(* Logix 5000 project; controller SPECK Emulate 5570 rev 30.12; software revision 30.00 *)

TASK MainTask (periodic, rate 5000 ms, priority 1, watchdog 5000 ms) : MainProgram

MODULES
   Local : Emulate 5570 (ICP 2, rev 30.12)
       : vendor 1 type 0 code 15 (ICP 0, rev 1.1, Output RPI 50 ms)
END_MODULES

TYPE UDT_BA :
STRUCT
   AL : BOOL;
END_STRUCT
END_TYPE

PROGRAM MainProgram   (* main routine MainRoutine *)
VAR
   SCAN_CYCLE_TIME : DINT;
   Speck_AS_res : DINT[2];
   Speck_AS_tmp : DINT;
   Speck_AS_X : DINT[2] := ([0] := -536870912);
   Speck_AS_Y : DINT[2] := ([0] := 1610612736);
   Speck_Block_size : DINT;
   Speck_Carry_Bit : DINT;
   Speck_Ciphertext : DINT[2,2];
   Speck_dec_i : DINT;
   Speck_dec_j : DINT;
   Speck_enc_i : DINT;
   Speck_enc_j : DINT;
   Speck_i : DINT;
   Speck_j : DINT;
   Speck_key_size : DINT;
   Speck_Plaintext : DINT[2,2];
   Speck_Rd_Max : DINT;
   Speck_Rotate_Result : DINT[2];
   Speck_Round_Keys : DINT[34,2];
   Speck_Sign_Bits : DINT[2];
   Speck_SR_m : DINT[2];
   Speck_tmp : DINT;
   Speck_tmp1 : DINT;
   Speck_Ver : DINT;
   Speck_x : DINT[2];
   Speck_y : DINT[2];
END_VAR

ROUTINE MainRoutine   (* ladder *)
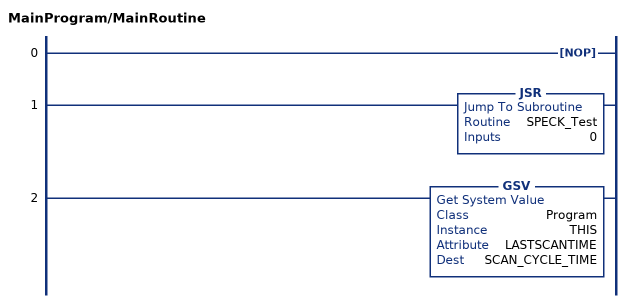
   0: NOP();
   1: JSR(SPECK_Test,0);
   2: GSV(Program,THIS,LASTSCANTIME,SCAN_CYCLE_TIME);
END_ROUTINE

ROUTINE SPECK_Add   (* structured text *)
   	//big addition low 32-bit
   		Speck_AS_res[0]:=0;
   		Speck_AS_res[1]:=0;
   		Speck_Sign_Bits[0].[0]:= Speck_AS_X[0].30; //keep the sign bit for big addition
   		Speck_Sign_Bits[0].[1]:= Speck_AS_X[0].31;
   		Speck_AS_X[0].31:=0;
   		Speck_AS_X[0].30:=0;
   
   		Speck_Sign_Bits[1].[0]:= Speck_AS_Y[0].30; //keep the sign bit for big addition
   		Speck_Sign_Bits[1].[1]:= Speck_AS_Y[0].31;
   		Speck_AS_Y[0].31:=0;
   		Speck_AS_Y[0].30:=0;
   
   		Speck_AS_res[0] := Speck_AS_X[0]+Speck_AS_Y[0];
   
   		Speck_Carry_Bit.[0]:= Speck_AS_res[0].30;
   
   		Speck_AS_tmp:=Speck_Sign_Bits[1]+Speck_Sign_Bits[0]+Speck_Carry_Bit;
   
   		Speck_AS_res[0].[30]:= Speck_AS_tmp.[0];
   		Speck_AS_res[0].[31]:= Speck_AS_tmp.[1];
   
   		Speck_Carry_Bit.[0]:= Speck_AS_tmp.[2];
   
   
   		Speck_AS_tmp:=0;
   		Speck_Sign_Bits[0]:=0;
   		Speck_Sign_Bits[1]:=0;
   
   //add high 32-bit
   if Speck_Ver>2 then
   		Speck_Sign_Bits[0].[0]:= Speck_AS_X[1].30; //keep the sign bit for big addition
   		Speck_Sign_Bits[0].[1]:= Speck_AS_X[1].31;
   		Speck_AS_X[1].31:=0;
   		Speck_AS_X[1].30:=0;
   
   		Speck_Sign_Bits[1].[0]:= Speck_AS_Y[1].30; //keep the sign bit for big addition
   		Speck_Sign_Bits[1].[1]:= Speck_AS_Y[1].31;
   		Speck_AS_Y[1].31:=0;
   		Speck_AS_Y[1].30:=0;
   
   		Speck_AS_res[1]:=Speck_AS_X[1]+Speck_AS_Y[1]+Speck_Carry_Bit;
   
   		Speck_Carry_Bit.[0]:= Speck_AS_res[1].30;
   
   		Speck_AS_tmp:=Speck_Sign_Bits[1]+Speck_Sign_Bits[0]+Speck_Carry_Bit;
   
   		Speck_AS_res[1].[30]:= Speck_AS_tmp.[0];
   		Speck_AS_res[1].[31]:= Speck_AS_tmp.[1];
   end_if;
   
   		//clear
   		Speck_Carry_Bit:=0;
   		Speck_AS_tmp:=0;
   		Speck_Sign_Bits[0]:=0;
   		Speck_Sign_Bits[1]:=0;
   		Speck_AS_X[0]:=0;
   		Speck_AS_X[1]:=0;
   		Speck_AS_Y[0]:=0;
   		Speck_AS_Y[1]:=0;
   
   
END_ROUTINE

ROUTINE SPECK_ClearKey   (* structured text *)
   
   Speck_Round_Keys[0,0]:=0;
   Speck_Round_Keys[1,0]:=0;
   Speck_Round_Keys[2,0]:=0;
   Speck_Round_Keys[3,0]:=0;
   Speck_Round_Keys[4,0]:=0;
   Speck_Round_Keys[5,0]:=0;
   Speck_Round_Keys[6,0]:=0;
   Speck_Round_Keys[7,0]:=0;
   Speck_Round_Keys[8,0]:=0;
   Speck_Round_Keys[9,0]:=0;
   Speck_Round_Keys[10,0]:=0;
   Speck_Round_Keys[11,0]:=0;
   Speck_Round_Keys[12,0]:=0;
   Speck_Round_Keys[13,0]:=0;
   Speck_Round_Keys[14,0]:=0;
   Speck_Round_Keys[15,0]:=0;
   Speck_Round_Keys[16,0]:=0;
   Speck_Round_Keys[17,0]:=0;
   Speck_Round_Keys[18,0]:=0;
   Speck_Round_Keys[19,0]:=0;
   Speck_Round_Keys[20,0]:=0;
   Speck_Round_Keys[21,0]:=0;
   Speck_Round_Keys[22,0]:=0;
   Speck_Round_Keys[23,0]:=0;
   Speck_Round_Keys[24,0]:=0;
   Speck_Round_Keys[25,0]:=0;
   Speck_Round_Keys[26,0]:=0;
END_ROUTINE

ROUTINE SPECK_Dec   (* structured text *)
   
   JSR(SPECK_Init);
   
   
   
   
   Case Speck_Ver Of
   
   0,1,2:
   	Speck_Plaintext[0,0]:=Speck_Ciphertext[0,0];
   	Speck_Plaintext[1,0]:=Speck_Ciphertext[1,0];
   
   	For Speck_i:=Speck_Rd_Max to 0 by -1 do
   
   		Speck_AS_res[0]:= Speck_Plaintext[1,0] XOR Speck_Plaintext[0,0];
   
   		Speck_SR_m[0]:=Speck_AS_res[0];
   		JSR(SPECK_Rotate_Right_Dec);      //rotate based on Speck_AS_res[0]
   
   		Speck_Plaintext[0,0]:= Speck_Rotate_Result[0];
   
   		Speck_AS_X[0]:= Speck_Plaintext[1,0] XOR Speck_Round_Keys[Speck_i,0];
   
   
   
   		if Speck_Ver=0 Then
   			Speck_AS_X[0].16:=1;
   			Speck_AS_res[0]:= (Speck_AS_X[0]- Speck_Plaintext[0,0]) AND 16#0000ffff; //??AND 16#ffff;
   		Else
   			Speck_AS_Y[0]:=Speck_Plaintext[0,0];
   			JSR(SPECK_Sub);
   		End_if;
   		Speck_SR_m[0]:=Speck_AS_res[0];
   		JSR(SPECK_Rotate_Left_Dec);      //rotate based on Speck_AS_res[0]
   		Speck_Plaintext[1,0]:=Speck_Rotate_Result[0];
   
   	End_for;
   
   3,4,5:
   	Speck_Plaintext[0,0]:=Speck_Ciphertext[0,0];
   	Speck_Plaintext[0,1]:=Speck_Ciphertext[0,1];
   	Speck_Plaintext[1,0]:=Speck_Ciphertext[1,0];
   	Speck_Plaintext[1,1]:=Speck_Ciphertext[1,1];
   
   	For Speck_i:=Speck_Rd_Max to 0 by -1 do
   
   		Speck_AS_res[0]:= Speck_Plaintext[0,0] XOR Speck_Plaintext[1,0];
   		Speck_AS_res[1]:= Speck_Plaintext[0,1] XOR Speck_Plaintext[1,1];
   
   
   		Speck_SR_m[0]:=Speck_AS_res[0];
   		Speck_SR_m[1]:=Speck_AS_res[1];
   		JSR(SPECK_Rotate_Right_Dec);      //rotate based on Speck_AS_res[0] and Speck_AS_res[1]
   
   		Speck_Plaintext[0,0]:= Speck_Rotate_Result[0];
   		Speck_Plaintext[0,1]:= Speck_Rotate_Result[1];
   
   		Speck_AS_X[0]:= Speck_Plaintext[1,0] XOR Speck_Round_Keys[Speck_i,0];
   		Speck_AS_X[1]:= Speck_Plaintext[1,1] XOR Speck_Round_Keys[Speck_i,1];
   
   
   		Speck_AS_Y[0]:=Speck_Plaintext[0,0];
   		Speck_AS_Y[1]:=Speck_Plaintext[0,1];
   		JSR(SPECK_Sub);
   
   		Speck_SR_m[0]:=Speck_AS_res[0];
   		Speck_SR_m[1]:=Speck_AS_res[1];
   		JSR(SPECK_Rotate_Left_Dec);      //rotate based on Speck_AS_res[0] and Speck_AS_res[1]
   		Speck_Plaintext[1,0]:=Speck_Rotate_Result[0];
   		Speck_Plaintext[1,1]:=Speck_Rotate_Result[1];
   	End_for;
   
   End_Case;
   
   
   
   
   
   
   JSR(SPECK_ClearKey);
   
   
   
   
   
   
   
   
END_ROUTINE

ROUTINE SPECK_Enc   (* structured text *)
   
   JSR(SPECK_Init);
   
   
   Case Speck_Ver Of
   
   0,1,2:
   	Speck_Ciphertext[0,0]:=Speck_Plaintext[0,0];
   	Speck_Ciphertext[1,0]:=Speck_Plaintext[1,0];
   
   	For Speck_i:=0 to Speck_Rd_Max by 1 do
   		Speck_SR_m[0]:=Speck_Ciphertext[1,0];
   		JSR(SPECK_Rotate_Right_Enc);       //c1>>>>
   
   		if Speck_Ver=0 Then
   			Speck_Ciphertext[1,0]:= (Speck_Rotate_Result[0] + Speck_Ciphertext[0,0]) XOR Speck_Round_Keys[Speck_i,0];
   			Speck_Ciphertext[1,0]:= Speck_Ciphertext[1,0] AND 16#0000ffff;
   		Else
   			Speck_AS_X[0]:=Speck_Rotate_Result[0];
   			Speck_AS_Y[0]:=Speck_Ciphertext[0,0];
   			JSR(SPECK_Add);
   			Speck_Ciphertext[1,0]:= Speck_AS_res[0] XOR Speck_Round_Keys[Speck_i,0];
   		End_if;
   
   
   		Speck_SR_m[0]:=Speck_Ciphertext[0,0];
   		JSR(SPECK_Rotate_Left_Enc);   //p0<<<
   		Speck_Ciphertext[0,0]:=Speck_Rotate_Result[0] XOR Speck_Ciphertext[1,0];
   	End_for;
   
   3,4,5:
   	Speck_Ciphertext[0,0]:=Speck_Plaintext[0,0];
   	Speck_Ciphertext[0,1]:=Speck_Plaintext[0,1];
   	Speck_Ciphertext[1,0]:=Speck_Plaintext[1,0];
   	Speck_Ciphertext[1,1]:=Speck_Plaintext[1,1];
   
   	For Speck_i:=0 to Speck_Rd_Max by 1 do
   		Speck_SR_m[0]:=Speck_Ciphertext[1,0];
   		Speck_SR_m[1]:=Speck_Ciphertext[1,1];
   		JSR(SPECK_Rotate_Right_Enc);       //c1>>>>
   
   		Speck_AS_X[0]:=Speck_Rotate_Result[0];
   		Speck_AS_X[1]:=Speck_Rotate_Result[1];
   		Speck_AS_Y[0]:=Speck_Ciphertext[0,0];
   		Speck_AS_Y[1]:=Speck_Ciphertext[0,1];
   		JSR(SPECK_Add);
   		Speck_Ciphertext[1,0]:= Speck_AS_res[0] XOR Speck_Round_Keys[Speck_i,0];
   	 	Speck_Ciphertext[1,1]:= Speck_AS_res[1] XOR Speck_Round_Keys[Speck_i,1];
   
   		Speck_SR_m[0]:=Speck_Ciphertext[0,0];
   		Speck_SR_m[1]:=Speck_Ciphertext[0,1];
   		JSR(SPECK_Rotate_Left_Enc);   //c0<<<
   		Speck_Ciphertext[0,0]:=Speck_Rotate_Result[0] XOR Speck_Ciphertext[1,0];
   		Speck_Ciphertext[0,1]:=Speck_Rotate_Result[1] XOR Speck_Ciphertext[1,1];
   	End_for;
   
   End_Case;
   
   
   JSR(SPECK_ClearKey);
   
   
   
   
   
   
END_ROUTINE

ROUTINE SPECK_Init   (* structured text *)
   CASE Speck_Ver Of
   	0:
   		//Speck_Rd_Max:=21;
   		Speck_Rd_Max:=21;
   		Speck_Round_Keys[0,0]:=256;
   		Speck_Round_Keys[1,0]:=5394;
   		Speck_Round_Keys[2,0]:=24957;
   		Speck_Round_Keys[3,0]:=5208;
   		Speck_Round_Keys[4,0]:=26905;
   		Speck_Round_Keys[5,0]:=30690;
   		Speck_Round_Keys[6,0]:=3209;
   		Speck_Round_Keys[7,0]:=52443;
   		Speck_Round_Keys[8,0]:=61418;
   		Speck_Round_Keys[9,0]:=20019;
   		Speck_Round_Keys[10,0]:=30452;
   		Speck_Round_Keys[11,0]:=22902;
   		Speck_Round_Keys[12,0]:=61067;
   		Speck_Round_Keys[13,0]:=56068;
   		Speck_Round_Keys[14,0]:=17943;
   		Speck_Round_Keys[15,0]:=62334;
   		Speck_Round_Keys[16,0]:=34740;
   		Speck_Round_Keys[17,0]:=36554;
   		Speck_Round_Keys[18,0]:=60827;
   		Speck_Round_Keys[19,0]:=14930;
   		Speck_Round_Keys[20,0]:=33321;
   		Speck_Round_Keys[21,0]:=60772;
   
   	1:
   		Speck_Rd_Max:=25;
   		Speck_Round_Keys[0,0]:=50462976;
   		Speck_Round_Keys[1,0]:=320668425;
   		Speck_Round_Keys[2,0]:=-1143468717;
   		Speck_Round_Keys[3,0]:=438530241;
   		Speck_Round_Keys[4,0]:=-463657251;
   		Speck_Round_Keys[5,0]:=1674264348;
   		Speck_Round_Keys[6,0]:=660176218;
   		Speck_Round_Keys[7,0]:=542209460;
   		Speck_Round_Keys[8,0]:=-620635233;
   		Speck_Round_Keys[9,0]:=-1743607096;
   		Speck_Round_Keys[10,0]:=377054067;
   		Speck_Round_Keys[11,0]:=-9280389;
   		Speck_Round_Keys[12,0]:=-858098844;
   		Speck_Round_Keys[13,0]:=-688605239;
   		Speck_Round_Keys[14,0]:=629784410;
   		Speck_Round_Keys[15,0]:=963910745;
   		Speck_Round_Keys[16,0]:=-2052674916;
   		Speck_Round_Keys[17,0]:=546222198;
   		Speck_Round_Keys[18,0]:=1906914590;
   		Speck_Round_Keys[19,0]:=-1895867933;
   		Speck_Round_Keys[20,0]:=1234172310;
   		Speck_Round_Keys[21,0]:=367819809;
   		Speck_Round_Keys[22,0]:=256446538;
   		Speck_Round_Keys[23,0]:=-655744580;
   		Speck_Round_Keys[24,0]:=-589610660;
   		Speck_Round_Keys[25,0]:=799533313;
   
   	2:
   		Speck_Rd_Max:=26;
   		Speck_Round_Keys[0,0]:=50462976;
   		Speck_Round_Keys[1,0]:=320668425;
   		Speck_Round_Keys[2,0]:=-1143468717;
   		Speck_Round_Keys[3,0]:=1696098252;
   		Speck_Round_Keys[4,0]:=1189104311;
   		Speck_Round_Keys[5,0]:=1426141042;
   		Speck_Round_Keys[6,0]:=246709480;
   		Speck_Round_Keys[7,0]:=-1769912550;
   		Speck_Round_Keys[8,0]:=-353799609;
   		Speck_Round_Keys[9,0]:=853261689;
   		Speck_Round_Keys[10,0]:=459475929;
   		Speck_Round_Keys[11,0]:=1977201121;
   		Speck_Round_Keys[12,0]:=317902096;
   		Speck_Round_Keys[13,0]:=-1273568388;
   		Speck_Round_Keys[14,0]:=2104671875;
   		Speck_Round_Keys[15,0]:=1924860368;
   		Speck_Round_Keys[16,0]:=-83442473;
   		Speck_Round_Keys[17,0]:=-1177375533;
   		Speck_Round_Keys[18,0]:=1274985820;
   		Speck_Round_Keys[19,0]:=-6786794;
   		Speck_Round_Keys[20,0]:=-1757815548;
   		Speck_Round_Keys[21,0]:=-512646929;
   		Speck_Round_Keys[22,0]:=-576779808;
   		Speck_Round_Keys[23,0]:=2113096485;
   		Speck_Round_Keys[24,0]:=-1495903407;
   		Speck_Round_Keys[25,0]:=1881079754;
   		Speck_Round_Keys[26,0]:=323482756;
   	3:
   		Speck_Rd_Max:=31;
   		Speck_Round_Keys[0,0]:=50462976;
   		Speck_Round_Keys[0,1]:=117835012;
   		Speck_Round_Keys[1,0]:=387777289;
   		Speck_Round_Keys[1,1]:=925186865;
   		Speck_Round_Keys[2,0]:=-1866200996;
   		Speck_Round_Keys[2,1]:=-115504692;
   		Speck_Round_Keys[3,0]:=1389131401;
   		Speck_Round_Keys[3,1]:=-961417096;
   		Speck_Round_Keys[4,0]:=-104671504;
   		Speck_Round_Keys[4,1]:=22007284;
   		Speck_Round_Keys[5,0]:=-31141930;
   		Speck_Round_Keys[5,1]:=-1241849372;
   		Speck_Round_Keys[6,0]:=-1334608642;
   		Speck_Round_Keys[6,1]:=-1553110700;
   		Speck_Round_Keys[7,0]:=-1607518733;
   		Speck_Round_Keys[7,1]:=-183408354;
   		Speck_Round_Keys[8,0]:=1512785245;
   		Speck_Round_Keys[8,1]:=1400155063;
   		Speck_Round_Keys[9,0]:=1306309285;
   		Speck_Round_Keys[9,1]:=-1915357664;
   		Speck_Round_Keys[10,0]:=-2036552680;
   		Speck_Round_Keys[10,1]:=-1304176695;
   		Speck_Round_Keys[11,0]:=1717585310;
   		Speck_Round_Keys[11,1]:=1967028860;
   		Speck_Round_Keys[12,0]:=-1515133381;
   		Speck_Round_Keys[12,1]:=2027309219;
   		Speck_Round_Keys[13,0]:=-876566318;
   		Speck_Round_Keys[13,1]:=-2028655837;
   		Speck_Round_Keys[14,0]:=1420015346;
   		Speck_Round_Keys[14,1]:=-1459647604;
   		Speck_Round_Keys[15,0]:=1135864441;
   		Speck_Round_Keys[15,1]:=1215544892;
   		Speck_Round_Keys[16,0]:=-1090139373;
   		Speck_Round_Keys[16,1]:=1998503932;
   		Speck_Round_Keys[17,0]:=629554464;
   		Speck_Round_Keys[17,1]:=-391725905;
   		Speck_Round_Keys[18,0]:=1548881043;
   		Speck_Round_Keys[18,1]:=-423433589;
   		Speck_Round_Keys[19,0]:=-1403906827;
   		Speck_Round_Keys[19,1]:=1299297729;
   		Speck_Round_Keys[20,0]:=623931612;
   		Speck_Round_Keys[20,1]:=-597642578;
   		Speck_Round_Keys[21,0]:=-503605439;
   		Speck_Round_Keys[21,1]:=-1340273989;
   		Speck_Round_Keys[22,0]:=-1558661814;
   		Speck_Round_Keys[22,1]:=-677874044;
   		Speck_Round_Keys[23,0]:=-436153575;
   		Speck_Round_Keys[23,1]:=-1574153598;
   		Speck_Round_Keys[24,0]:=-1107754936;
   		Speck_Round_Keys[24,1]:=-534129026;
   		Speck_Round_Keys[25,0]:=-934347329;
   		Speck_Round_Keys[25,1]:=1733661236;
   		Speck_Round_Keys[26,0]:=-889099940;
   		Speck_Round_Keys[26,1]:=1696021744;
   		Speck_Round_Keys[27,0]:=2038535449;
   		Speck_Round_Keys[27,1]:=617553688;
   		Speck_Round_Keys[28,0]:=-609241302;
   		Speck_Round_Keys[28,1]:=950234834;
   		Speck_Round_Keys[29,0]:=834331396;
   		Speck_Round_Keys[29,1]:=-556188418;
   		Speck_Round_Keys[30,0]:=393261669;
   		Speck_Round_Keys[30,1]:=-985851719;
   		Speck_Round_Keys[31,0]:=-611399361;
   		Speck_Round_Keys[31,1]:=563726448;
   
   	4:
   		Speck_Rd_Max:=32;
   		Speck_Round_Keys[0,0]:=50462976;
   		Speck_Round_Keys[0,1]:=117835012;
   		Speck_Round_Keys[1,0]:=387777289;
   		Speck_Round_Keys[1,1]:=925186865;
   		Speck_Round_Keys[2,0]:=-1814557358;
   		Speck_Round_Keys[2,1]:=-32143154;
   		Speck_Round_Keys[3,0]:=975663304;
   		Speck_Round_Keys[3,1]:=-142025835;
   		Speck_Round_Keys[4,0]:=1365845657;
   		Speck_Round_Keys[4,1]:=-1365849265;
   		Speck_Round_Keys[5,0]:=-1203291782;
   		Speck_Round_Keys[5,1]:=2032907671;
   		Speck_Round_Keys[6,0]:=1560168396;
   		Speck_Round_Keys[6,1]:=-1637668590;
   		Speck_Round_Keys[7,0]:=-1379701829;
   		Speck_Round_Keys[7,1]:=-1503031408;
   		Speck_Round_Keys[8,0]:=863596189;
   		Speck_Round_Keys[8,1]:=-158551405;
   		Speck_Round_Keys[9,0]:=-1375147243;
   		Speck_Round_Keys[9,1]:=1636284355;
   		Speck_Round_Keys[10,0]:=-1272900118;
   		Speck_Round_Keys[10,1]:=-1368340852;
   		Speck_Round_Keys[11,0]:=-1352763690;
   		Speck_Round_Keys[11,1]:=-624911147;
   		Speck_Round_Keys[12,0]:=1003580318;
   		Speck_Round_Keys[12,1]:=-899281693;
   		Speck_Round_Keys[13,0]:=894738061;
   		Speck_Round_Keys[13,1]:=490681490;
   		Speck_Round_Keys[14,0]:=691090703;
   		Speck_Round_Keys[14,1]:=-1398656019;
   		Speck_Round_Keys[15,0]:=-57361246;
   		Speck_Round_Keys[15,1]:=1122098217;
   		Speck_Round_Keys[16,0]:=-1648511106;
   		Speck_Round_Keys[16,1]:=-1121331570;
   		Speck_Round_Keys[17,0]:=866086775;
   		Speck_Round_Keys[17,1]:=1964995237;
   		Speck_Round_Keys[18,0]:=1776548963;
   		Speck_Round_Keys[18,1]:=1228016885;
   		Speck_Round_Keys[19,0]:=1960676415;
   		Speck_Round_Keys[19,1]:=-2107754217;
   		Speck_Round_Keys[20,0]:=-146881239;
   		Speck_Round_Keys[20,1]:=1236388362;
   		Speck_Round_Keys[21,0]:=176991942;
   		Speck_Round_Keys[21,1]:=586401854;
   		Speck_Round_Keys[22,0]:=-272894130;
   		Speck_Round_Keys[22,1]:=-271496784;
   		Speck_Round_Keys[23,0]:=615566260;
   		Speck_Round_Keys[23,1]:=46828238;
   		Speck_Round_Keys[24,0]:=1089140610;
   		Speck_Round_Keys[24,1]:=-1802072153;
   		Speck_Round_Keys[25,0]:=-1928078593;
   		Speck_Round_Keys[25,1]:=-56185516;
   		Speck_Round_Keys[26,0]:=199725135;
   		Speck_Round_Keys[26,1]:=-98821494;
   		Speck_Round_Keys[27,0]:=625825488;
   		Speck_Round_Keys[27,1]:=898955530;
   		Speck_Round_Keys[28,0]:=2044356237;
   		Speck_Round_Keys[28,1]:=1226041899;
   		Speck_Round_Keys[29,0]:=445115415;
   		Speck_Round_Keys[29,1]:=-1335488765;
   		Speck_Round_Keys[30,0]:=1088748615;
   		Speck_Round_Keys[30,1]:=1048296253;
   		Speck_Round_Keys[31,0]:=-1633766600;
   		Speck_Round_Keys[31,1]:=1336503665;
   		Speck_Round_Keys[32,0]:=818288393;
   		Speck_Round_Keys[32,1]:=925749944;
   
   	5:
   		Speck_Rd_Max:=33;
   		Speck_Round_Keys[0,0]:=50462976;
   		Speck_Round_Keys[0,1]:=117835012;
   		Speck_Round_Keys[1,0]:=387777289;
   		Speck_Round_Keys[1,1]:=925186865;
   		Speck_Round_Keys[2,0]:=-1814557358;
   		Speck_Round_Keys[2,1]:=-32143154;
   		Speck_Round_Keys[3,0]:=825445886;
   		Speck_Round_Keys[3,1]:=-426188641;
   		Speck_Round_Keys[4,0]:=-875023107;
   		Speck_Round_Keys[4,1]:=-614403765;
   		Speck_Round_Keys[5,0]:=1287832312;
   		Speck_Round_Keys[5,1]:=766486467;
   		Speck_Round_Keys[6,0]:=1583653339;
   		Speck_Round_Keys[6,1]:=-71769488;
   		Speck_Round_Keys[7,0]:=-477893905;
   		Speck_Round_Keys[7,1]:=-613443100;
   		Speck_Round_Keys[8,0]:=-1668630227;
   		Speck_Round_Keys[8,1]:=689605941;
   		Speck_Round_Keys[9,0]:=-493428094;
   		Speck_Round_Keys[9,1]:=191183550;
   		Speck_Round_Keys[10,0]:=1544592767;
   		Speck_Round_Keys[10,1]:=1614952126;
   		Speck_Round_Keys[11,0]:=-1911170916;
   		Speck_Round_Keys[11,1]:=-1239078670;
   		Speck_Round_Keys[12,0]:=-793616599;
   		Speck_Round_Keys[12,1]:=272735697;
   		Speck_Round_Keys[13,0]:=-1670774794;
   		Speck_Round_Keys[13,1]:=-42866885;
   		Speck_Round_Keys[14,0]:=2140630675;
   		Speck_Round_Keys[14,1]:=-1901518332;
   		Speck_Round_Keys[15,0]:=965541820;
   		Speck_Round_Keys[15,1]:=771988221;
   		Speck_Round_Keys[16,0]:=583075628;
   		Speck_Round_Keys[16,1]:=-1667248145;
   		Speck_Round_Keys[17,0]:=-313137463;
   		Speck_Round_Keys[17,1]:=637176179;
   		Speck_Round_Keys[18,0]:=-1498142708;
   		Speck_Round_Keys[18,1]:=1770100833;
   		Speck_Round_Keys[19,0]:=-1744597129;
   		Speck_Round_Keys[19,1]:=2070075508;
   		Speck_Round_Keys[20,0]:=1659016958;
   		Speck_Round_Keys[20,1]:=-231399730;
   		Speck_Round_Keys[21,0]:=1991902719;
   		Speck_Round_Keys[21,1]:=-1496087855;
   		Speck_Round_Keys[22,0]:=1169655590;
   		Speck_Round_Keys[22,1]:=-1919490457;
   		Speck_Round_Keys[23,0]:=-1645822159;
   		Speck_Round_Keys[23,1]:=-1099482754;
   		Speck_Round_Keys[24,0]:=-1350724487;
   		Speck_Round_Keys[24,1]:=890732295;
   		Speck_Round_Keys[25,0]:=-410951696;
   		Speck_Round_Keys[25,1]:=-1201049147;
   		Speck_Round_Keys[26,0]:=272319978;
   		Speck_Round_Keys[26,1]:=2104999935;
   		Speck_Round_Keys[27,0]:=-2103336674;
   		Speck_Round_Keys[27,1]:=-1719430836;
   		Speck_Round_Keys[28,0]:=1848838133;
   		Speck_Round_Keys[28,1]:=512289202;
   		Speck_Round_Keys[29,0]:=1338443291;
   		Speck_Round_Keys[29,1]:=2046847095;
   		Speck_Round_Keys[30,0]:=2113057135;
   		Speck_Round_Keys[30,1]:=393340252;
   		Speck_Round_Keys[31,0]:=-1141349352;
   		Speck_Round_Keys[31,1]:=-1563733213;
   		Speck_Round_Keys[32,0]:=2146821003;
   		Speck_Round_Keys[32,1]:=1073939284;
   		Speck_Round_Keys[33,0]:=-1705594250;
   		Speck_Round_Keys[33,1]:=-187535528;
   End_CASE;
   
END_ROUTINE

ROUTINE SPECK_Rotate_Left_Dec   (* structured text *)
   Speck_Rotate_Result[0]:=0;
   Speck_Rotate_Result[1]:=0;
   
   CASE Speck_Ver Of
   	0:
   		Speck_Rotate_Result[0].[6]:=Speck_SR_m[0].[15];
   		Speck_Rotate_Result[0].[5]:=Speck_SR_m[0].[14];
   		Speck_Rotate_Result[0].[4]:=Speck_SR_m[0].[13];
   		Speck_Rotate_Result[0].[3]:=Speck_SR_m[0].[12];
   		Speck_Rotate_Result[0].[2]:=Speck_SR_m[0].[11];
   		Speck_Rotate_Result[0].[1]:=Speck_SR_m[0].[10];
   		Speck_Rotate_Result[0].[0]:=Speck_SR_m[0].[9];
   		Speck_Rotate_Result[0].[15]:=Speck_SR_m[0].[8];
   		Speck_Rotate_Result[0].[14]:=Speck_SR_m[0].[7];
   		Speck_Rotate_Result[0].[13]:=Speck_SR_m[0].[6];
   		Speck_Rotate_Result[0].[12]:=Speck_SR_m[0].[5];
   		Speck_Rotate_Result[0].[11]:=Speck_SR_m[0].[4];
   		Speck_Rotate_Result[0].[10]:=Speck_SR_m[0].[3];
   		Speck_Rotate_Result[0].[9]:=Speck_SR_m[0].[2];
   		Speck_Rotate_Result[0].[8]:=Speck_SR_m[0].[1];
   		Speck_Rotate_Result[0].[7]:=Speck_SR_m[0].[0];
   	1,2:
   		Speck_Rotate_Result[0].[7]:=Speck_SR_m[0].[31];
   		Speck_Rotate_Result[0].[6]:=Speck_SR_m[0].[30];
   		Speck_Rotate_Result[0].[5]:=Speck_SR_m[0].[29];
   		Speck_Rotate_Result[0].[4]:=Speck_SR_m[0].[28];
   		Speck_Rotate_Result[0].[3]:=Speck_SR_m[0].[27];
   		Speck_Rotate_Result[0].[2]:=Speck_SR_m[0].[26];
   		Speck_Rotate_Result[0].[1]:=Speck_SR_m[0].[25];
   		Speck_Rotate_Result[0].[0]:=Speck_SR_m[0].[24];
   		Speck_Rotate_Result[0].[31]:=Speck_SR_m[0].[23];
   		Speck_Rotate_Result[0].[30]:=Speck_SR_m[0].[22];
   		Speck_Rotate_Result[0].[29]:=Speck_SR_m[0].[21];
   		Speck_Rotate_Result[0].[28]:=Speck_SR_m[0].[20];
   		Speck_Rotate_Result[0].[27]:=Speck_SR_m[0].[19];
   		Speck_Rotate_Result[0].[26]:=Speck_SR_m[0].[18];
   		Speck_Rotate_Result[0].[25]:=Speck_SR_m[0].[17];
   		Speck_Rotate_Result[0].[24]:=Speck_SR_m[0].[16];
   		Speck_Rotate_Result[0].[23]:=Speck_SR_m[0].[15];
   		Speck_Rotate_Result[0].[22]:=Speck_SR_m[0].[14];
   		Speck_Rotate_Result[0].[21]:=Speck_SR_m[0].[13];
   		Speck_Rotate_Result[0].[20]:=Speck_SR_m[0].[12];
   		Speck_Rotate_Result[0].[19]:=Speck_SR_m[0].[11];
   		Speck_Rotate_Result[0].[18]:=Speck_SR_m[0].[10];
   		Speck_Rotate_Result[0].[17]:=Speck_SR_m[0].[9];
   		Speck_Rotate_Result[0].[16]:=Speck_SR_m[0].[8];
   		Speck_Rotate_Result[0].[15]:=Speck_SR_m[0].[7];
   		Speck_Rotate_Result[0].[14]:=Speck_SR_m[0].[6];
   		Speck_Rotate_Result[0].[13]:=Speck_SR_m[0].[5];
   		Speck_Rotate_Result[0].[12]:=Speck_SR_m[0].[4];
   		Speck_Rotate_Result[0].[11]:=Speck_SR_m[0].[3];
   		Speck_Rotate_Result[0].[10]:=Speck_SR_m[0].[2];
   		Speck_Rotate_Result[0].[9]:=Speck_SR_m[0].[1];
   		Speck_Rotate_Result[0].[8]:=Speck_SR_m[0].[0];
   	3,4,5:
   		Speck_Rotate_Result[0].[7]:=Speck_SR_m[1].[31];
   		Speck_Rotate_Result[0].[6]:=Speck_SR_m[1].[30];
   		Speck_Rotate_Result[0].[5]:=Speck_SR_m[1].[29];
   		Speck_Rotate_Result[0].[4]:=Speck_SR_m[1].[28];
   		Speck_Rotate_Result[0].[3]:=Speck_SR_m[1].[27];
   		Speck_Rotate_Result[0].[2]:=Speck_SR_m[1].[26];
   		Speck_Rotate_Result[0].[1]:=Speck_SR_m[1].[25];
   		Speck_Rotate_Result[0].[0]:=Speck_SR_m[1].[24];
   		Speck_Rotate_Result[1].[31]:=Speck_SR_m[1].[23];
   		Speck_Rotate_Result[1].[30]:=Speck_SR_m[1].[22];
   		Speck_Rotate_Result[1].[29]:=Speck_SR_m[1].[21];
   		Speck_Rotate_Result[1].[28]:=Speck_SR_m[1].[20];
   		Speck_Rotate_Result[1].[27]:=Speck_SR_m[1].[19];
   		Speck_Rotate_Result[1].[26]:=Speck_SR_m[1].[18];
   		Speck_Rotate_Result[1].[25]:=Speck_SR_m[1].[17];
   		Speck_Rotate_Result[1].[24]:=Speck_SR_m[1].[16];
   		Speck_Rotate_Result[1].[23]:=Speck_SR_m[1].[15];
   		Speck_Rotate_Result[1].[22]:=Speck_SR_m[1].[14];
   		Speck_Rotate_Result[1].[21]:=Speck_SR_m[1].[13];
   		Speck_Rotate_Result[1].[20]:=Speck_SR_m[1].[12];
   		Speck_Rotate_Result[1].[19]:=Speck_SR_m[1].[11];
   		Speck_Rotate_Result[1].[18]:=Speck_SR_m[1].[10];
   		Speck_Rotate_Result[1].[17]:=Speck_SR_m[1].[9];
   		Speck_Rotate_Result[1].[16]:=Speck_SR_m[1].[8];
   		Speck_Rotate_Result[1].[15]:=Speck_SR_m[1].[7];
   		Speck_Rotate_Result[1].[14]:=Speck_SR_m[1].[6];
   		Speck_Rotate_Result[1].[13]:=Speck_SR_m[1].[5];
   		Speck_Rotate_Result[1].[12]:=Speck_SR_m[1].[4];
   		Speck_Rotate_Result[1].[11]:=Speck_SR_m[1].[3];
   		Speck_Rotate_Result[1].[10]:=Speck_SR_m[1].[2];
   		Speck_Rotate_Result[1].[9]:=Speck_SR_m[1].[1];
   		Speck_Rotate_Result[1].[8]:=Speck_SR_m[1].[0];
   		Speck_Rotate_Result[1].[7]:=Speck_SR_m[0].[31];
   		Speck_Rotate_Result[1].[6]:=Speck_SR_m[0].[30];
   		Speck_Rotate_Result[1].[5]:=Speck_SR_m[0].[29];
   		Speck_Rotate_Result[1].[4]:=Speck_SR_m[0].[28];
   		Speck_Rotate_Result[1].[3]:=Speck_SR_m[0].[27];
   		Speck_Rotate_Result[1].[2]:=Speck_SR_m[0].[26];
   		Speck_Rotate_Result[1].[1]:=Speck_SR_m[0].[25];
   		Speck_Rotate_Result[1].[0]:=Speck_SR_m[0].[24];
   		Speck_Rotate_Result[0].[31]:=Speck_SR_m[0].[23];
   		Speck_Rotate_Result[0].[30]:=Speck_SR_m[0].[22];
   		Speck_Rotate_Result[0].[29]:=Speck_SR_m[0].[21];
   		Speck_Rotate_Result[0].[28]:=Speck_SR_m[0].[20];
   		Speck_Rotate_Result[0].[27]:=Speck_SR_m[0].[19];
   		Speck_Rotate_Result[0].[26]:=Speck_SR_m[0].[18];
   		Speck_Rotate_Result[0].[25]:=Speck_SR_m[0].[17];
   		Speck_Rotate_Result[0].[24]:=Speck_SR_m[0].[16];
   		Speck_Rotate_Result[0].[23]:=Speck_SR_m[0].[15];
   		Speck_Rotate_Result[0].[22]:=Speck_SR_m[0].[14];
   		Speck_Rotate_Result[0].[21]:=Speck_SR_m[0].[13];
   		Speck_Rotate_Result[0].[20]:=Speck_SR_m[0].[12];
   		Speck_Rotate_Result[0].[19]:=Speck_SR_m[0].[11];
   		Speck_Rotate_Result[0].[18]:=Speck_SR_m[0].[10];
   		Speck_Rotate_Result[0].[17]:=Speck_SR_m[0].[9];
   		Speck_Rotate_Result[0].[16]:=Speck_SR_m[0].[8];
   		Speck_Rotate_Result[0].[15]:=Speck_SR_m[0].[7];
   		Speck_Rotate_Result[0].[14]:=Speck_SR_m[0].[6];
   		Speck_Rotate_Result[0].[13]:=Speck_SR_m[0].[5];
   		Speck_Rotate_Result[0].[12]:=Speck_SR_m[0].[4];
   		Speck_Rotate_Result[0].[11]:=Speck_SR_m[0].[3];
   		Speck_Rotate_Result[0].[10]:=Speck_SR_m[0].[2];
   		Speck_Rotate_Result[0].[9]:=Speck_SR_m[0].[1];
   		Speck_Rotate_Result[0].[8]:=Speck_SR_m[0].[0];
   End_CASE;
   
END_ROUTINE

ROUTINE SPECK_Rotate_Left_Enc   (* structured text *)
   Speck_Rotate_Result[0]:=0;
   Speck_Rotate_Result[1]:=0;
   CASE Speck_Ver Of
   	0:
   		Speck_Rotate_Result[0].[1]:=Speck_SR_m[0].[15];
   		Speck_Rotate_Result[0].[0]:=Speck_SR_m[0].[14];
   		Speck_Rotate_Result[0].[15]:=Speck_SR_m[0].[13];
   		Speck_Rotate_Result[0].[14]:=Speck_SR_m[0].[12];
   		Speck_Rotate_Result[0].[13]:=Speck_SR_m[0].[11];
   		Speck_Rotate_Result[0].[12]:=Speck_SR_m[0].[10];
   		Speck_Rotate_Result[0].[11]:=Speck_SR_m[0].[9];
   		Speck_Rotate_Result[0].[10]:=Speck_SR_m[0].[8];
   		Speck_Rotate_Result[0].[9]:=Speck_SR_m[0].[7];
   		Speck_Rotate_Result[0].[8]:=Speck_SR_m[0].[6];
   		Speck_Rotate_Result[0].[7]:=Speck_SR_m[0].[5];
   		Speck_Rotate_Result[0].[6]:=Speck_SR_m[0].[4];
   		Speck_Rotate_Result[0].[5]:=Speck_SR_m[0].[3];
   		Speck_Rotate_Result[0].[4]:=Speck_SR_m[0].[2];
   		Speck_Rotate_Result[0].[3]:=Speck_SR_m[0].[1];
   		Speck_Rotate_Result[0].[2]:=Speck_SR_m[0].[0];
   	1,2:
   		Speck_Rotate_Result[0].[2]:=Speck_SR_m[0].[31];
   		Speck_Rotate_Result[0].[1]:=Speck_SR_m[0].[30];
   		Speck_Rotate_Result[0].[0]:=Speck_SR_m[0].[29];
   		Speck_Rotate_Result[0].[31]:=Speck_SR_m[0].[28];
   		Speck_Rotate_Result[0].[30]:=Speck_SR_m[0].[27];
   		Speck_Rotate_Result[0].[29]:=Speck_SR_m[0].[26];
   		Speck_Rotate_Result[0].[28]:=Speck_SR_m[0].[25];
   		Speck_Rotate_Result[0].[27]:=Speck_SR_m[0].[24];
   		Speck_Rotate_Result[0].[26]:=Speck_SR_m[0].[23];
   		Speck_Rotate_Result[0].[25]:=Speck_SR_m[0].[22];
   		Speck_Rotate_Result[0].[24]:=Speck_SR_m[0].[21];
   		Speck_Rotate_Result[0].[23]:=Speck_SR_m[0].[20];
   		Speck_Rotate_Result[0].[22]:=Speck_SR_m[0].[19];
   		Speck_Rotate_Result[0].[21]:=Speck_SR_m[0].[18];
   		Speck_Rotate_Result[0].[20]:=Speck_SR_m[0].[17];
   		Speck_Rotate_Result[0].[19]:=Speck_SR_m[0].[16];
   		Speck_Rotate_Result[0].[18]:=Speck_SR_m[0].[15];
   		Speck_Rotate_Result[0].[17]:=Speck_SR_m[0].[14];
   		Speck_Rotate_Result[0].[16]:=Speck_SR_m[0].[13];
   		Speck_Rotate_Result[0].[15]:=Speck_SR_m[0].[12];
   		Speck_Rotate_Result[0].[14]:=Speck_SR_m[0].[11];
   		Speck_Rotate_Result[0].[13]:=Speck_SR_m[0].[10];
   		Speck_Rotate_Result[0].[12]:=Speck_SR_m[0].[9];
   		Speck_Rotate_Result[0].[11]:=Speck_SR_m[0].[8];
   		Speck_Rotate_Result[0].[10]:=Speck_SR_m[0].[7];
   		Speck_Rotate_Result[0].[9]:=Speck_SR_m[0].[6];
   		Speck_Rotate_Result[0].[8]:=Speck_SR_m[0].[5];
   		Speck_Rotate_Result[0].[7]:=Speck_SR_m[0].[4];
   		Speck_Rotate_Result[0].[6]:=Speck_SR_m[0].[3];
   		Speck_Rotate_Result[0].[5]:=Speck_SR_m[0].[2];
   		Speck_Rotate_Result[0].[4]:=Speck_SR_m[0].[1];
   		Speck_Rotate_Result[0].[3]:=Speck_SR_m[0].[0];
   	3,4,5:
   		Speck_Rotate_Result[0].[2]:=Speck_SR_m[1].[31];
   		Speck_Rotate_Result[0].[1]:=Speck_SR_m[1].[30];
   		Speck_Rotate_Result[0].[0]:=Speck_SR_m[1].[29];
   		Speck_Rotate_Result[1].[31]:=Speck_SR_m[1].[28];
   		Speck_Rotate_Result[1].[30]:=Speck_SR_m[1].[27];
   		Speck_Rotate_Result[1].[29]:=Speck_SR_m[1].[26];
   		Speck_Rotate_Result[1].[28]:=Speck_SR_m[1].[25];
   		Speck_Rotate_Result[1].[27]:=Speck_SR_m[1].[24];
   		Speck_Rotate_Result[1].[26]:=Speck_SR_m[1].[23];
   		Speck_Rotate_Result[1].[25]:=Speck_SR_m[1].[22];
   		Speck_Rotate_Result[1].[24]:=Speck_SR_m[1].[21];
   		Speck_Rotate_Result[1].[23]:=Speck_SR_m[1].[20];
   		Speck_Rotate_Result[1].[22]:=Speck_SR_m[1].[19];
   		Speck_Rotate_Result[1].[21]:=Speck_SR_m[1].[18];
   		Speck_Rotate_Result[1].[20]:=Speck_SR_m[1].[17];
   		Speck_Rotate_Result[1].[19]:=Speck_SR_m[1].[16];
   		Speck_Rotate_Result[1].[18]:=Speck_SR_m[1].[15];
   		Speck_Rotate_Result[1].[17]:=Speck_SR_m[1].[14];
   		Speck_Rotate_Result[1].[16]:=Speck_SR_m[1].[13];
   		Speck_Rotate_Result[1].[15]:=Speck_SR_m[1].[12];
   		Speck_Rotate_Result[1].[14]:=Speck_SR_m[1].[11];
   		Speck_Rotate_Result[1].[13]:=Speck_SR_m[1].[10];
   		Speck_Rotate_Result[1].[12]:=Speck_SR_m[1].[9];
   		Speck_Rotate_Result[1].[11]:=Speck_SR_m[1].[8];
   		Speck_Rotate_Result[1].[10]:=Speck_SR_m[1].[7];
   		Speck_Rotate_Result[1].[9]:=Speck_SR_m[1].[6];
   		Speck_Rotate_Result[1].[8]:=Speck_SR_m[1].[5];
   		Speck_Rotate_Result[1].[7]:=Speck_SR_m[1].[4];
   		Speck_Rotate_Result[1].[6]:=Speck_SR_m[1].[3];
   		Speck_Rotate_Result[1].[5]:=Speck_SR_m[1].[2];
   		Speck_Rotate_Result[1].[4]:=Speck_SR_m[1].[1];
   		Speck_Rotate_Result[1].[3]:=Speck_SR_m[1].[0];
   		Speck_Rotate_Result[1].[2]:=Speck_SR_m[0].[31];
   		Speck_Rotate_Result[1].[1]:=Speck_SR_m[0].[30];
   		Speck_Rotate_Result[1].[0]:=Speck_SR_m[0].[29];
   		Speck_Rotate_Result[0].[31]:=Speck_SR_m[0].[28];
   		Speck_Rotate_Result[0].[30]:=Speck_SR_m[0].[27];
   		Speck_Rotate_Result[0].[29]:=Speck_SR_m[0].[26];
   		Speck_Rotate_Result[0].[28]:=Speck_SR_m[0].[25];
   		Speck_Rotate_Result[0].[27]:=Speck_SR_m[0].[24];
   		Speck_Rotate_Result[0].[26]:=Speck_SR_m[0].[23];
   		Speck_Rotate_Result[0].[25]:=Speck_SR_m[0].[22];
   		Speck_Rotate_Result[0].[24]:=Speck_SR_m[0].[21];
   		Speck_Rotate_Result[0].[23]:=Speck_SR_m[0].[20];
   		Speck_Rotate_Result[0].[22]:=Speck_SR_m[0].[19];
   		Speck_Rotate_Result[0].[21]:=Speck_SR_m[0].[18];
   		Speck_Rotate_Result[0].[20]:=Speck_SR_m[0].[17];
   		Speck_Rotate_Result[0].[19]:=Speck_SR_m[0].[16];
   		Speck_Rotate_Result[0].[18]:=Speck_SR_m[0].[15];
   		Speck_Rotate_Result[0].[17]:=Speck_SR_m[0].[14];
   		Speck_Rotate_Result[0].[16]:=Speck_SR_m[0].[13];
   		Speck_Rotate_Result[0].[15]:=Speck_SR_m[0].[12];
   		Speck_Rotate_Result[0].[14]:=Speck_SR_m[0].[11];
   		Speck_Rotate_Result[0].[13]:=Speck_SR_m[0].[10];
   		Speck_Rotate_Result[0].[12]:=Speck_SR_m[0].[9];
   		Speck_Rotate_Result[0].[11]:=Speck_SR_m[0].[8];
   		Speck_Rotate_Result[0].[10]:=Speck_SR_m[0].[7];
   		Speck_Rotate_Result[0].[9]:=Speck_SR_m[0].[6];
   		Speck_Rotate_Result[0].[8]:=Speck_SR_m[0].[5];
   		Speck_Rotate_Result[0].[7]:=Speck_SR_m[0].[4];
   		Speck_Rotate_Result[0].[6]:=Speck_SR_m[0].[3];
   		Speck_Rotate_Result[0].[5]:=Speck_SR_m[0].[2];
   		Speck_Rotate_Result[0].[4]:=Speck_SR_m[0].[1];
   		Speck_Rotate_Result[0].[3]:=Speck_SR_m[0].[0];
   End_CASE;
   
END_ROUTINE

ROUTINE SPECK_Rotate_Right_Dec   (* structured text *)
   Speck_Rotate_Result[0]:=0;
   Speck_Rotate_Result[1]:=0;
   
   CASE Speck_Ver Of
   	0:
   		Speck_Rotate_Result[0].[13]:=Speck_SR_m[0].[15];
   		Speck_Rotate_Result[0].[12]:=Speck_SR_m[0].[14];
   		Speck_Rotate_Result[0].[11]:=Speck_SR_m[0].[13];
   		Speck_Rotate_Result[0].[10]:=Speck_SR_m[0].[12];
   		Speck_Rotate_Result[0].[9]:=Speck_SR_m[0].[11];
   		Speck_Rotate_Result[0].[8]:=Speck_SR_m[0].[10];
   		Speck_Rotate_Result[0].[7]:=Speck_SR_m[0].[9];
   		Speck_Rotate_Result[0].[6]:=Speck_SR_m[0].[8];
   		Speck_Rotate_Result[0].[5]:=Speck_SR_m[0].[7];
   		Speck_Rotate_Result[0].[4]:=Speck_SR_m[0].[6];
   		Speck_Rotate_Result[0].[3]:=Speck_SR_m[0].[5];
   		Speck_Rotate_Result[0].[2]:=Speck_SR_m[0].[4];
   		Speck_Rotate_Result[0].[1]:=Speck_SR_m[0].[3];
   		Speck_Rotate_Result[0].[0]:=Speck_SR_m[0].[2];
   		Speck_Rotate_Result[0].[15]:=Speck_SR_m[0].[1];
   		Speck_Rotate_Result[0].[14]:=Speck_SR_m[0].[0];
   	1,2:
   		Speck_Rotate_Result[0].[28]:=Speck_SR_m[0].[31];
   		Speck_Rotate_Result[0].[27]:=Speck_SR_m[0].[30];
   		Speck_Rotate_Result[0].[26]:=Speck_SR_m[0].[29];
   		Speck_Rotate_Result[0].[25]:=Speck_SR_m[0].[28];
   		Speck_Rotate_Result[0].[24]:=Speck_SR_m[0].[27];
   		Speck_Rotate_Result[0].[23]:=Speck_SR_m[0].[26];
   		Speck_Rotate_Result[0].[22]:=Speck_SR_m[0].[25];
   		Speck_Rotate_Result[0].[21]:=Speck_SR_m[0].[24];
   		Speck_Rotate_Result[0].[20]:=Speck_SR_m[0].[23];
   		Speck_Rotate_Result[0].[19]:=Speck_SR_m[0].[22];
   		Speck_Rotate_Result[0].[18]:=Speck_SR_m[0].[21];
   		Speck_Rotate_Result[0].[17]:=Speck_SR_m[0].[20];
   		Speck_Rotate_Result[0].[16]:=Speck_SR_m[0].[19];
   		Speck_Rotate_Result[0].[15]:=Speck_SR_m[0].[18];
   		Speck_Rotate_Result[0].[14]:=Speck_SR_m[0].[17];
   		Speck_Rotate_Result[0].[13]:=Speck_SR_m[0].[16];
   		Speck_Rotate_Result[0].[12]:=Speck_SR_m[0].[15];
   		Speck_Rotate_Result[0].[11]:=Speck_SR_m[0].[14];
   		Speck_Rotate_Result[0].[10]:=Speck_SR_m[0].[13];
   		Speck_Rotate_Result[0].[9]:=Speck_SR_m[0].[12];
   		Speck_Rotate_Result[0].[8]:=Speck_SR_m[0].[11];
   		Speck_Rotate_Result[0].[7]:=Speck_SR_m[0].[10];
   		Speck_Rotate_Result[0].[6]:=Speck_SR_m[0].[9];
   		Speck_Rotate_Result[0].[5]:=Speck_SR_m[0].[8];
   		Speck_Rotate_Result[0].[4]:=Speck_SR_m[0].[7];
   		Speck_Rotate_Result[0].[3]:=Speck_SR_m[0].[6];
   		Speck_Rotate_Result[0].[2]:=Speck_SR_m[0].[5];
   		Speck_Rotate_Result[0].[1]:=Speck_SR_m[0].[4];
   		Speck_Rotate_Result[0].[0]:=Speck_SR_m[0].[3];
   		Speck_Rotate_Result[0].[31]:=Speck_SR_m[0].[2];
   		Speck_Rotate_Result[0].[30]:=Speck_SR_m[0].[1];
   		Speck_Rotate_Result[0].[29]:=Speck_SR_m[0].[0];
   	3,4,5:
   		Speck_Rotate_Result[1].[28]:=Speck_SR_m[1].[31];
   		Speck_Rotate_Result[1].[27]:=Speck_SR_m[1].[30];
   		Speck_Rotate_Result[1].[26]:=Speck_SR_m[1].[29];
   		Speck_Rotate_Result[1].[25]:=Speck_SR_m[1].[28];
   		Speck_Rotate_Result[1].[24]:=Speck_SR_m[1].[27];
   		Speck_Rotate_Result[1].[23]:=Speck_SR_m[1].[26];
   		Speck_Rotate_Result[1].[22]:=Speck_SR_m[1].[25];
   		Speck_Rotate_Result[1].[21]:=Speck_SR_m[1].[24];
   		Speck_Rotate_Result[1].[20]:=Speck_SR_m[1].[23];
   		Speck_Rotate_Result[1].[19]:=Speck_SR_m[1].[22];
   		Speck_Rotate_Result[1].[18]:=Speck_SR_m[1].[21];
   		Speck_Rotate_Result[1].[17]:=Speck_SR_m[1].[20];
   		Speck_Rotate_Result[1].[16]:=Speck_SR_m[1].[19];
   		Speck_Rotate_Result[1].[15]:=Speck_SR_m[1].[18];
   		Speck_Rotate_Result[1].[14]:=Speck_SR_m[1].[17];
   		Speck_Rotate_Result[1].[13]:=Speck_SR_m[1].[16];
   		Speck_Rotate_Result[1].[12]:=Speck_SR_m[1].[15];
   		Speck_Rotate_Result[1].[11]:=Speck_SR_m[1].[14];
   		Speck_Rotate_Result[1].[10]:=Speck_SR_m[1].[13];
   		Speck_Rotate_Result[1].[9]:=Speck_SR_m[1].[12];
   		Speck_Rotate_Result[1].[8]:=Speck_SR_m[1].[11];
   		Speck_Rotate_Result[1].[7]:=Speck_SR_m[1].[10];
   		Speck_Rotate_Result[1].[6]:=Speck_SR_m[1].[9];
   		Speck_Rotate_Result[1].[5]:=Speck_SR_m[1].[8];
   		Speck_Rotate_Result[1].[4]:=Speck_SR_m[1].[7];
   		Speck_Rotate_Result[1].[3]:=Speck_SR_m[1].[6];
   		Speck_Rotate_Result[1].[2]:=Speck_SR_m[1].[5];
   		Speck_Rotate_Result[1].[1]:=Speck_SR_m[1].[4];
   		Speck_Rotate_Result[1].[0]:=Speck_SR_m[1].[3];
   		Speck_Rotate_Result[0].[31]:=Speck_SR_m[1].[2];
   		Speck_Rotate_Result[0].[30]:=Speck_SR_m[1].[1];
   		Speck_Rotate_Result[0].[29]:=Speck_SR_m[1].[0];
   		Speck_Rotate_Result[0].[28]:=Speck_SR_m[0].[31];
   		Speck_Rotate_Result[0].[27]:=Speck_SR_m[0].[30];
   		Speck_Rotate_Result[0].[26]:=Speck_SR_m[0].[29];
   		Speck_Rotate_Result[0].[25]:=Speck_SR_m[0].[28];
   		Speck_Rotate_Result[0].[24]:=Speck_SR_m[0].[27];
   		Speck_Rotate_Result[0].[23]:=Speck_SR_m[0].[26];
   		Speck_Rotate_Result[0].[22]:=Speck_SR_m[0].[25];
   		Speck_Rotate_Result[0].[21]:=Speck_SR_m[0].[24];
   		Speck_Rotate_Result[0].[20]:=Speck_SR_m[0].[23];
   		Speck_Rotate_Result[0].[19]:=Speck_SR_m[0].[22];
   		Speck_Rotate_Result[0].[18]:=Speck_SR_m[0].[21];
   		Speck_Rotate_Result[0].[17]:=Speck_SR_m[0].[20];
   		Speck_Rotate_Result[0].[16]:=Speck_SR_m[0].[19];
   		Speck_Rotate_Result[0].[15]:=Speck_SR_m[0].[18];
   		Speck_Rotate_Result[0].[14]:=Speck_SR_m[0].[17];
   		Speck_Rotate_Result[0].[13]:=Speck_SR_m[0].[16];
   		Speck_Rotate_Result[0].[12]:=Speck_SR_m[0].[15];
   		Speck_Rotate_Result[0].[11]:=Speck_SR_m[0].[14];
   		Speck_Rotate_Result[0].[10]:=Speck_SR_m[0].[13];
   		Speck_Rotate_Result[0].[9]:=Speck_SR_m[0].[12];
   		Speck_Rotate_Result[0].[8]:=Speck_SR_m[0].[11];
   		Speck_Rotate_Result[0].[7]:=Speck_SR_m[0].[10];
   		Speck_Rotate_Result[0].[6]:=Speck_SR_m[0].[9];
   		Speck_Rotate_Result[0].[5]:=Speck_SR_m[0].[8];
   		Speck_Rotate_Result[0].[4]:=Speck_SR_m[0].[7];
   		Speck_Rotate_Result[0].[3]:=Speck_SR_m[0].[6];
   		Speck_Rotate_Result[0].[2]:=Speck_SR_m[0].[5];
   		Speck_Rotate_Result[0].[1]:=Speck_SR_m[0].[4];
   		Speck_Rotate_Result[0].[0]:=Speck_SR_m[0].[3];
   		Speck_Rotate_Result[1].[31]:=Speck_SR_m[0].[2];
   		Speck_Rotate_Result[1].[30]:=Speck_SR_m[0].[1];
   		Speck_Rotate_Result[1].[29]:=Speck_SR_m[0].[0];
   End_CASE;
   
END_ROUTINE

ROUTINE SPECK_Rotate_Right_Enc   (* structured text *)
   Speck_Rotate_Result[0]:=0;
   Speck_Rotate_Result[1]:=0;
   
   CASE Speck_Ver Of
   	0:
   		Speck_Rotate_Result[0].[8]:=Speck_SR_m[0].[15];
   		Speck_Rotate_Result[0].[7]:=Speck_SR_m[0].[14];
   		Speck_Rotate_Result[0].[6]:=Speck_SR_m[0].[13];
   		Speck_Rotate_Result[0].[5]:=Speck_SR_m[0].[12];
   		Speck_Rotate_Result[0].[4]:=Speck_SR_m[0].[11];
   		Speck_Rotate_Result[0].[3]:=Speck_SR_m[0].[10];
   		Speck_Rotate_Result[0].[2]:=Speck_SR_m[0].[9];
   		Speck_Rotate_Result[0].[1]:=Speck_SR_m[0].[8];
   		Speck_Rotate_Result[0].[0]:=Speck_SR_m[0].[7];
   		Speck_Rotate_Result[0].[15]:=Speck_SR_m[0].[6];
   		Speck_Rotate_Result[0].[14]:=Speck_SR_m[0].[5];
   		Speck_Rotate_Result[0].[13]:=Speck_SR_m[0].[4];
   		Speck_Rotate_Result[0].[12]:=Speck_SR_m[0].[3];
   		Speck_Rotate_Result[0].[11]:=Speck_SR_m[0].[2];
   		Speck_Rotate_Result[0].[10]:=Speck_SR_m[0].[1];
   		Speck_Rotate_Result[0].[9]:=Speck_SR_m[0].[0];
   	1,2:
   		Speck_Rotate_Result[0].[23]:=Speck_SR_m[0].[31];
   		Speck_Rotate_Result[0].[22]:=Speck_SR_m[0].[30];
   		Speck_Rotate_Result[0].[21]:=Speck_SR_m[0].[29];
   		Speck_Rotate_Result[0].[20]:=Speck_SR_m[0].[28];
   		Speck_Rotate_Result[0].[19]:=Speck_SR_m[0].[27];
   		Speck_Rotate_Result[0].[18]:=Speck_SR_m[0].[26];
   		Speck_Rotate_Result[0].[17]:=Speck_SR_m[0].[25];
   		Speck_Rotate_Result[0].[16]:=Speck_SR_m[0].[24];
   		Speck_Rotate_Result[0].[15]:=Speck_SR_m[0].[23];
   		Speck_Rotate_Result[0].[14]:=Speck_SR_m[0].[22];
   		Speck_Rotate_Result[0].[13]:=Speck_SR_m[0].[21];
   		Speck_Rotate_Result[0].[12]:=Speck_SR_m[0].[20];
   		Speck_Rotate_Result[0].[11]:=Speck_SR_m[0].[19];
   		Speck_Rotate_Result[0].[10]:=Speck_SR_m[0].[18];
   		Speck_Rotate_Result[0].[9]:=Speck_SR_m[0].[17];
   		Speck_Rotate_Result[0].[8]:=Speck_SR_m[0].[16];
   		Speck_Rotate_Result[0].[7]:=Speck_SR_m[0].[15];
   		Speck_Rotate_Result[0].[6]:=Speck_SR_m[0].[14];
   		Speck_Rotate_Result[0].[5]:=Speck_SR_m[0].[13];
   		Speck_Rotate_Result[0].[4]:=Speck_SR_m[0].[12];
   		Speck_Rotate_Result[0].[3]:=Speck_SR_m[0].[11];
   		Speck_Rotate_Result[0].[2]:=Speck_SR_m[0].[10];
   		Speck_Rotate_Result[0].[1]:=Speck_SR_m[0].[9];
   		Speck_Rotate_Result[0].[0]:=Speck_SR_m[0].[8];
   		Speck_Rotate_Result[0].[31]:=Speck_SR_m[0].[7];
   		Speck_Rotate_Result[0].[30]:=Speck_SR_m[0].[6];
   		Speck_Rotate_Result[0].[29]:=Speck_SR_m[0].[5];
   		Speck_Rotate_Result[0].[28]:=Speck_SR_m[0].[4];
   		Speck_Rotate_Result[0].[27]:=Speck_SR_m[0].[3];
   		Speck_Rotate_Result[0].[26]:=Speck_SR_m[0].[2];
   		Speck_Rotate_Result[0].[25]:=Speck_SR_m[0].[1];
   		Speck_Rotate_Result[0].[24]:=Speck_SR_m[0].[0];
   	3,4,5:
   		Speck_Rotate_Result[1].[23]:=Speck_SR_m[1].[31];
   		Speck_Rotate_Result[1].[22]:=Speck_SR_m[1].[30];
   		Speck_Rotate_Result[1].[21]:=Speck_SR_m[1].[29];
   		Speck_Rotate_Result[1].[20]:=Speck_SR_m[1].[28];
   		Speck_Rotate_Result[1].[19]:=Speck_SR_m[1].[27];
   		Speck_Rotate_Result[1].[18]:=Speck_SR_m[1].[26];
   		Speck_Rotate_Result[1].[17]:=Speck_SR_m[1].[25];
   		Speck_Rotate_Result[1].[16]:=Speck_SR_m[1].[24];
   		Speck_Rotate_Result[1].[15]:=Speck_SR_m[1].[23];
   		Speck_Rotate_Result[1].[14]:=Speck_SR_m[1].[22];
   		Speck_Rotate_Result[1].[13]:=Speck_SR_m[1].[21];
   		Speck_Rotate_Result[1].[12]:=Speck_SR_m[1].[20];
   		Speck_Rotate_Result[1].[11]:=Speck_SR_m[1].[19];
   		Speck_Rotate_Result[1].[10]:=Speck_SR_m[1].[18];
   		Speck_Rotate_Result[1].[9]:=Speck_SR_m[1].[17];
   		Speck_Rotate_Result[1].[8]:=Speck_SR_m[1].[16];
   		Speck_Rotate_Result[1].[7]:=Speck_SR_m[1].[15];
   		Speck_Rotate_Result[1].[6]:=Speck_SR_m[1].[14];
   		Speck_Rotate_Result[1].[5]:=Speck_SR_m[1].[13];
   		Speck_Rotate_Result[1].[4]:=Speck_SR_m[1].[12];
   		Speck_Rotate_Result[1].[3]:=Speck_SR_m[1].[11];
   		Speck_Rotate_Result[1].[2]:=Speck_SR_m[1].[10];
   		Speck_Rotate_Result[1].[1]:=Speck_SR_m[1].[9];
   		Speck_Rotate_Result[1].[0]:=Speck_SR_m[1].[8];
   		Speck_Rotate_Result[0].[31]:=Speck_SR_m[1].[7];
   		Speck_Rotate_Result[0].[30]:=Speck_SR_m[1].[6];
   		Speck_Rotate_Result[0].[29]:=Speck_SR_m[1].[5];
   		Speck_Rotate_Result[0].[28]:=Speck_SR_m[1].[4];
   		Speck_Rotate_Result[0].[27]:=Speck_SR_m[1].[3];
   		Speck_Rotate_Result[0].[26]:=Speck_SR_m[1].[2];
   		Speck_Rotate_Result[0].[25]:=Speck_SR_m[1].[1];
   		Speck_Rotate_Result[0].[24]:=Speck_SR_m[1].[0];
   		Speck_Rotate_Result[0].[23]:=Speck_SR_m[0].[31];
   		Speck_Rotate_Result[0].[22]:=Speck_SR_m[0].[30];
   		Speck_Rotate_Result[0].[21]:=Speck_SR_m[0].[29];
   		Speck_Rotate_Result[0].[20]:=Speck_SR_m[0].[28];
   		Speck_Rotate_Result[0].[19]:=Speck_SR_m[0].[27];
   		Speck_Rotate_Result[0].[18]:=Speck_SR_m[0].[26];
   		Speck_Rotate_Result[0].[17]:=Speck_SR_m[0].[25];
   		Speck_Rotate_Result[0].[16]:=Speck_SR_m[0].[24];
   		Speck_Rotate_Result[0].[15]:=Speck_SR_m[0].[23];
   		Speck_Rotate_Result[0].[14]:=Speck_SR_m[0].[22];
   		Speck_Rotate_Result[0].[13]:=Speck_SR_m[0].[21];
   		Speck_Rotate_Result[0].[12]:=Speck_SR_m[0].[20];
   		Speck_Rotate_Result[0].[11]:=Speck_SR_m[0].[19];
   		Speck_Rotate_Result[0].[10]:=Speck_SR_m[0].[18];
   		Speck_Rotate_Result[0].[9]:=Speck_SR_m[0].[17];
   		Speck_Rotate_Result[0].[8]:=Speck_SR_m[0].[16];
   		Speck_Rotate_Result[0].[7]:=Speck_SR_m[0].[15];
   		Speck_Rotate_Result[0].[6]:=Speck_SR_m[0].[14];
   		Speck_Rotate_Result[0].[5]:=Speck_SR_m[0].[13];
   		Speck_Rotate_Result[0].[4]:=Speck_SR_m[0].[12];
   		Speck_Rotate_Result[0].[3]:=Speck_SR_m[0].[11];
   		Speck_Rotate_Result[0].[2]:=Speck_SR_m[0].[10];
   		Speck_Rotate_Result[0].[1]:=Speck_SR_m[0].[9];
   		Speck_Rotate_Result[0].[0]:=Speck_SR_m[0].[8];
   		Speck_Rotate_Result[1].[31]:=Speck_SR_m[0].[7];
   		Speck_Rotate_Result[1].[30]:=Speck_SR_m[0].[6];
   		Speck_Rotate_Result[1].[29]:=Speck_SR_m[0].[5];
   		Speck_Rotate_Result[1].[28]:=Speck_SR_m[0].[4];
   		Speck_Rotate_Result[1].[27]:=Speck_SR_m[0].[3];
   		Speck_Rotate_Result[1].[26]:=Speck_SR_m[0].[2];
   		Speck_Rotate_Result[1].[25]:=Speck_SR_m[0].[1];
   		Speck_Rotate_Result[1].[24]:=Speck_SR_m[0].[0];
   End_CASE;
   
END_ROUTINE

ROUTINE SPECK_Sub   (* structured text *)
   Speck_AS_res[0]:=0;
   Speck_AS_res[1]:=0;
   
   	//big substraction low-32-bit
   		Speck_Sign_Bits[0].[0]:= Speck_AS_X[0].29; //keep the sign bit for big addition
   		Speck_Sign_Bits[0].[1]:= Speck_AS_X[0].30; //keep the sign bit for big addition
   		Speck_Sign_Bits[0].[2]:= Speck_AS_X[0].31; //keep the sign bit for big addition
   
   		Speck_AS_X[0].29:=0;
   		Speck_AS_X[0].30 :=1;   //give x  a 'virtual' borrow bit
   		Speck_AS_X[0].31:=0;
   
   
   
   		Speck_Sign_Bits[1].[0]:= Speck_AS_Y[0].29;
   		Speck_Sign_Bits[1].[1]:= Speck_AS_Y[0].30; //keep the sign bit for big addition
   		Speck_Sign_Bits[1].[2]:= Speck_AS_Y[0].31;
   		Speck_AS_Y[0].31:=0;
   		Speck_AS_Y[0].30:=0;
   		Speck_AS_Y[0].29:=0;
   
   		Speck_AS_res[0] := Speck_AS_X[0]-Speck_AS_Y[0];
   
   		Speck_Carry_Bit.[0]:= NOT Speck_AS_res[0].30;
   
   		Speck_Sign_Bits[0].[4]:=1;  //to ensure that Sign_Bits[0]> Sign_Bits[1]
   		Speck_AS_tmp:=Speck_Sign_Bits[0]-Speck_Sign_Bits[1]-Speck_Carry_Bit;
   
   
   
   		Speck_Carry_Bit.[0] := Speck_AS_tmp.[3];
   		Speck_AS_res[0].29:= Speck_AS_tmp.[0];
   		Speck_AS_res[0].30:= Speck_AS_tmp.[1];
   		Speck_AS_res[0].31:= Speck_AS_tmp.[2];
   
   
   		Speck_AS_tmp:=0;
   	 	Speck_Sign_Bits[0]:=0;
   	 	Speck_Sign_Bits[1]:=0;
   
   If Speck_Ver>2 Then
   
   		//sub high 32-bit
   
   		Speck_Sign_Bits[0].[0]:= Speck_AS_X[1].29; //keep the sign bit for big addition
   		Speck_Sign_Bits[0].[1]:= Speck_AS_X[1].30; //keep the sign bit for big addition
   		Speck_Sign_Bits[0].[2]:= Speck_AS_X[1].31; //keep the sign bit for big addition
   
   		Speck_AS_X[1].29:=0;
   		Speck_AS_X[1].30 :=1;   //give x  a 'virtual' borrow bit
   		Speck_AS_X[1].31:=0;
   
   
   
   		Speck_Sign_Bits[1].[0]:= Speck_AS_Y[1].29;
   		Speck_Sign_Bits[1].[1]:= Speck_AS_Y[1].30; //keep the sign bit for big addition
   		Speck_Sign_Bits[1].[2]:= Speck_AS_Y[1].31;
   		Speck_AS_Y[1].31:=0;
   		Speck_AS_Y[1].30:=0;
   		Speck_AS_Y[1].29:=0;
   
   		Speck_AS_res[1] := Speck_AS_X[1]-Speck_AS_Y[1] -Speck_Carry_Bit;
   
   		Speck_Carry_Bit.[0]:= NOT Speck_AS_res[1].30;
   
   		Speck_Sign_Bits[0].[4]:=1;
   		Speck_AS_tmp:=Speck_Sign_Bits[0]-Speck_Sign_Bits[1]-Speck_Carry_Bit;
   
   
   
   		Speck_AS_res[1].29:= Speck_AS_tmp.[0];
   		Speck_AS_res[1].30:= Speck_AS_tmp.[1];
   		Speck_AS_res[1].31:= Speck_AS_tmp.[2];
   
   End_If;
   
   
   		//clear
   		Speck_Carry_Bit:=0;
   		Speck_AS_tmp:=0;
   		Speck_Sign_Bits[0]:=0;
   		Speck_Sign_Bits[1]:=0;
   		Speck_AS_X[0]:=0;
   		Speck_AS_X[1]:=0;
   		Speck_AS_Y[0]:=0;
   		Speck_AS_Y[1]:=0;
   
END_ROUTINE

ROUTINE SPECK_Test   (* structured text *)
   if S:FS then
   	Speck_Ver:=3;     // 0: 32/64, 1: 64: 96, 2: 64:128, 3:128/128, 4:128/192, 5: 128/256
   	//32-64
   	Case Speck_Ver Of
   		0,1,2:
   			//Speck_Plaintext[0,0]:=16#694c; //Upper bits of current plaintext
   			//Speck_Plaintext[1,0]:=16#6574;  //Lower bits of current plaintext
   			//Speck_Plaintext[0,0]:=1936613733; //Upper bits of current plaintext
   			//Speck_Plaintext[1,0]:=1952532000;  //Lower bits of current plaintext
   			Speck_Plaintext[0,0]:=1953841965; //Upper bits of current plaintext
   			Speck_Plaintext[1,0]:=997352820;  //Lower bits of current plaintext
   
   		3,4,5:
   			Speck_Plaintext[0,0]:=1684106528; //Upper bits of current plaintext
   			Speck_Plaintext[0,1]:=1953046629;//Lower bits of current plaintext
   			Speck_Plaintext[1,0]:=1970365728; //Upper bits of current plaintext
   			Speck_Plaintext[1,1]:=1818326633; //Lower bits of current plaintext
   (*
   			Speck_Plaintext[0,0]:=544501349;  //ver=4
   			Speck_Plaintext[0,1]:=1126199156;
   			Speck_Plaintext[1,0]:=1717922152;
   			Speck_Plaintext[1,1]:=1918978080;*)
   
   (*
   			Speck_Plaintext[0,0]:=1852796784; //ver=5
   			Speck_Plaintext[0,1]:=539914853;
   			Speck_Plaintext[1,0]:=1948282441;
   			Speck_Plaintext[1,1]:=1702063976;*)
   	End_Case;
   	JSR(SPECK_Enc);
   	//JSR(SPECK_Dec);
   end_if;
   
   
   	//JSR(SPECK_Dec);
   
   
   
   (*
   
   Speck_Ver:=3;
   Speck_AS_Y[0]:=-536872146;
   Speck_AS_Y[1]:=-536872146;
   Speck_AS_X[0]:=1610625810;
   Speck_AS_X[1]:=1610625810;
   
   
   JSR(SPECK_Add);
   
   
   Speck_AS_X[0]:=Speck_AS_res[0];
   Speck_AS_X[1]:=Speck_AS_res[1];
   
   Speck_AS_Y[0]:=-536872146;
   Speck_AS_Y[1]:=-536872146;
   
   
   JSR(SPECK_Sub);
   
   *)
   
   
   
   
   
   
   
   
   
   
   
END_ROUTINE
END_PROGRAM
